INTERFACE I_PositionalDrive EXTENDS I_Drive

PROPERTY ABSTRACT CurrentPosition : LREAL
GET
END_GET
SET
END_SET
END_PROPERTY

METHOD ABSTRACT moveAbsolute : BOOL
VAR_INPUT
	newTarget : LREAL; 
END_VAR
END_METHOD

METHOD ABSTRACT moveRelative : BOOL
VAR_INPUT
	distance : LREAL;
END_VAR
END_METHOD

PROPERTY ABSTRACT TargetPosition : LREAL
GET
END_GET
SET
END_SET
END_PROPERTY

END_INTERFACE

(* stored: Version 1.1.0.1, ProductVersion 3.1.4024.11
   Itf I_PositionalDrive: Id {d3b144fb-f698-482d-9db8-649a39fe9d24}
   Folder Properties: Id {cacec72b-3d1f-47b7-abce-48f3a22265b6}
   Property CurrentPosition: Id {163278cf-f135-4311-a280-19e0fc73602d}
   Get Get: Id {f03c1c00-6590-4c8c-8593-fdc94541d64f}
   Set Set: Id {e50a4420-ba8d-4bf4-b8ef-6ae90ef0b70b}
   Method moveAbsolute: Id {4fb3220a-9ea1-4f96-b8de-0af48986a4b5}
   Method moveRelative: Id {413f6949-f6bb-4630-8086-ac8d20c9f65b}
   Property TargetPosition: Id {d76f5395-76cf-4061-8c77-336d3eb2b4ee}
   Get Get: Id {8bf52deb-a2de-4e21-a783-cda9e1127e79}
   Set Set: Id {87cf6527-f222-482b-881b-0b571918624d} *)
